# B&R Automation Studio project TestAsProj
Automation Studio 4.12.2.93; Project for testing the OpcUaUnitTesting Python script; technology packages: mappView 5.19.0

## Configuration ARSim

CPU PC_any, AutomationRuntime B4.93, Build 4.1.2, Vc 

### Task classes (Cpu.sw)
```
Cyclic#1 (cycle 10000 us, tolerance 0 us):
  BasicTest <- BasicTest.prg
Cyclic#2 (cycle 20000 us, tolerance 20000 us):
  GetInfo <- GetInfo.prg
Binaries: udbdef, mvLoader, FWRules, OpcUaSrv, TCData, sysconf, Role, User, iomap, ashwd, asfw, arconfig, ashwac
Libraries: arssl, fileio, AsARCfg, runtime, AsBrStr
```

### Hardware
```
PC : PC_any v1.1.1.0 (OrderNumber=PC)
  Connector IF3:
    InternetAddress = 172.27.224.1
  ConfigurationID = TestAsProj_ARSim
  Cyclic1Duration = 10000
  Cyclic1Tolerance = 0
  Cyclic2Duration = 20000
  Cyclic2Tolerance = 20000
  FileDevice1
  FileDeviceName1 = USER
  FileDevicePath1 = USER_PATH
  ActivateOpcUa = 1
  OpcUaInformationModels_PV_Version = 1
```

### Config.mpaudittrail - PC/mappServices/Config.mpaudittrail
```
Element gAuditTrail (Type=mpaudittrail)
  Audit:
    Events:
      [0] = 16
      [1] = 19
    TextSource = TXT
      OutputFormat = MpAudit/Event/Root
    Export:
      Encrypt = FALSE
  Alarms = MpAlarmX
```

### Config_1.mpalarmxcore - PC/mappServices/Config_1.mpalarmxcore
```
Element gAlarmXCore (Type=mpalarmxcore)
```

## Logical view

Binary libraries used (declarations not repeated): operator, runtime, astime, AsIecCon, AsBrStr, AsARCfg

### Global.typ - Global data types
```iecst
TYPE
	GlobalTestStruct : 	STRUCT
		TestUDINT : UDINT;
		TestBOOL : BOOL;
		TestSTRING : STRING[50];
		TestSubStruct : GlobalTestSubStruct;
	END_STRUCT;
	GlobalTestSubStruct : 	STRUCT
		TestREAL : REAL;
		TestLREAL : LREAL;
	END_STRUCT;
END_TYPE
```

### Global.var - Global variables
```iecst
VAR
	gGlobalInt : INT := -100;
	gGlobalUInt : UINT := 100;
	gGlobalString : STRING[50] := 'Test String?!';
	gTestStruct : GlobalTestStruct := (TestUDINT:=45678,TestBOOL:=TRUE,TestSTRING:='Test String 2',TestSubStruct:=(TestREAL:=123.4,TestLREAL:=432.1));
END_VAR
```

### Package Logical/Libraries - Global libraries

- Visualisation Logical/mappView (not shown)

### Program Logical/GetInfo (IEC)

#### Types.typ
```iecst
TYPE
	VisInfo_type : 	STRUCT
		IpAddr : STRING[80];
		NumConnectedClients : USINT;
		IsItFriday : STRING[10];
	END_STRUCT;
	InfoRefreshState_enum :
		(
		INFO_REFRESH_STATE_WAIT,
		INFO_REFRESH_STATE_GET_IP,
		INFO_REFRESH_STATE_GET_DAY,
		INFO_REFRESH_STATE_ERROR
		);
END_TYPE
```

#### Variables.var
```iecst
VAR
	VisInfo : VisInfo_type;
	InfoRefreshState : InfoRefreshState_enum;
	CmdRefreshInfo : BOOL;
	CmdErrorReset : BOOL;
	Error : BOOL;
	DtStruct : DTStructure;
END_VAR
(*Function Blocks*)
VAR
	fb_CfgGetIpAddr : CfgGetIPAddr;
	fb_DTStructureGetTime : DTStructureGetTime;
END_VAR
```

#### Main.st
```iecst
PROGRAM _INIT
    CmdRefreshInfo := TRUE;

END_PROGRAM

PROGRAM _CYCLIC
    CASE InfoRefreshState OF
        INFO_REFRESH_STATE_WAIT:
            IF CmdRefreshInfo THEN
                CmdRefreshInfo := FALSE;
                InfoRefreshState := INFO_REFRESH_STATE_GET_IP;
            END_IF;

        INFO_REFRESH_STATE_GET_IP:
            fb_CfgGetIpAddr.enable := TRUE;
            fb_CfgGetIpAddr.pDevice := ADR('IF3');
            fb_CfgGetIpAddr.pIPAddr := ADR(VisInfo.IpAddr);
            fb_CfgGetIpAddr.Len := SIZEOF(VisInfo.IpAddr);

            IF (fb_CfgGetIpAddr.status <> ERR_FUB_BUSY) AND (fb_CfgGetIpAddr.status <> ERR_FUB_ENABLE_FALSE) THEN
                IF fb_CfgGetIpAddr.status = ERR_OK THEN
                    fb_CfgGetIpAddr.enable := FALSE;
                    InfoRefreshState := INFO_REFRESH_STATE_GET_DAY;
                ELSE
                    Error := TRUE;
                    InfoRefreshState := INFO_REFRESH_STATE_ERROR;
                END_IF;
            END_IF;

        INFO_REFRESH_STATE_GET_DAY:
            brsmemset(ADR(VisInfo.IsItFriday), 0, SIZEOF(VisInfo.IsItFriday));
            brsstrcpy(ADR(VisInfo.IsItFriday), ADR('No :('));

            fb_DTStructureGetTime.enable := TRUE;
            fb_DTStructureGetTime.pDTStructure := ADR(DtStruct);

            IF (fb_DTStructureGetTime.status <> ERR_FUB_BUSY) AND (fb_DTStructureGetTime.status <> ERR_FUB_ENABLE_FALSE) THEN
                IF fb_DTStructureGetTime.status = ERR_OK THEN
                    fb_DTStructureGetTime.enable := FALSE;
                    IF DtStruct.wday = 5 THEN
                        brsmemset(ADR(VisInfo.IsItFriday), 0, SIZEOF(VisInfo.IsItFriday));
                        brsstrcpy(ADR(VisInfo.IsItFriday), ADR('Yes!'));
                    END_IF;
                    InfoRefreshState := INFO_REFRESH_STATE_WAIT;
                ELSE
                    Error := TRUE;
                    InfoRefreshState := INFO_REFRESH_STATE_ERROR;
                END_IF;
            END_IF;

        INFO_REFRESH_STATE_ERROR:
            IF CmdErrorReset THEN
                CmdErrorReset := FALSE;
                Error := FALSE;
                fb_CfgGetIpAddr.enable := FALSE;
                InfoRefreshState := INFO_REFRESH_STATE_WAIT;
            END_IF;

    END_CASE;

    //Call function blocks
    fb_CfgGetIpAddr();
    fb_DTStructureGetTime();
END_PROGRAM
```

### Program Logical/BasicTest (IEC)

#### Variables.var
```iecst
VAR
	TestBOOL : BOOL := TRUE;
	TestDINT : DINT := 65534;
	TestDT : DATE_AND_TIME;
	TestTIME : TIME := T#1d;
	AdditionIn1 : REAL;
	AdditionIn2 : REAL;
	AdditionOut : REAL;
END_VAR
```

#### Main.st
```iecst
PROGRAM _INIT
    gGlobalInt;
    gGlobalUInt;
    gGlobalString;
    gTestStruct;

    TestBOOL;
    TestDINT;
    TestDT;
    TestTIME;

END_PROGRAM

PROGRAM _CYCLIC
	AdditionOut := AdditionIn1 + AdditionIn2;

END_PROGRAM
```

### Program Logical/Alarms

#### Variables.var
```iecst
VAR
	fb_MpAlarmXCore : MpAlarmXCore;
END_VAR
```

#### Main.st
```iecst
PROGRAM _INIT
    fb_MpAlarmXCore.MpLink := ADR(gAlarmXCore);
    fb_MpAlarmXCore.Enable := TRUE;

END_PROGRAM

PROGRAM _CYCLIC
	fb_MpAlarmXCore();

END_PROGRAM

PROGRAM _EXIT
	fb_MpAlarmXCore(Enable := FALSE);

END_PROGRAM
```

### Program Logical/Audit

#### Variables.var
```iecst
VAR
	fb_MpAuditTrail : MpAuditTrail;
END_VAR
```

#### Main.st
```iecst
PROGRAM _INIT
    fb_MpAuditTrail.MpLink := ADR(gAuditTrail);
    fb_MpAuditTrail.Enable := TRUE;
    fb_MpAuditTrail.DeviceName := ADR('FD_Audit');

END_PROGRAM

PROGRAM _CYCLIC
	fb_MpAuditTrail();

END_PROGRAM

PROGRAM _EXIT
	fb_MpAuditTrail(Enable := FALSE);

END_PROGRAM
```

### Program Logical/WaterHeat

#### Main.st
```iecst
PROGRAM _INIT
    // Initial values
    WaterTemperature := BASE_TEMPERATURE;
    WaterLevel := 0.0;

    HeatRate := 0.3;
    CoolRate := 0.1;
    FillRate := 1.0;
    DrainRate := 1.0;

END_PROGRAM

PROGRAM _CYCLIC
	// Heating
    IF HeaterOn THEN
        WaterTemperature := WaterTemperature + (HeatRate/CYCLES_PER_SECOND);
    ELSE
        WaterTemperature := WaterTemperature - (CoolRate/CYCLES_PER_SECOND);
    END_IF;

    IF WaterTemperature > MAX_TEMPERATURE THEN
        WaterTemperature := MAX_TEMPERATURE;
    ELSIF WaterTemperature < BASE_TEMPERATURE THEN
        WaterTemperature := BASE_TEMPERATURE;
    END_IF;

    // Filling and Draining
    IF FillValveOpen THEN
        WaterLevel := WaterLevel + (FillRate/CYCLES_PER_SECOND);
    END_IF;

    IF DrainValveOpen THEN
        WaterLevel := WaterLevel - (DrainRate/CYCLES_PER_SECOND);
    END_IF;

    IF WaterLevel > MAX_LEVEL THEN
        WaterLevel := MAX_LEVEL;
        FillValveOpen := FALSE;
    ELSIF WaterLevel < MIN_LEVEL THEN
        WaterLevel := MIN_LEVEL;
        DrainValveOpen := FALSE;
    END_IF;

END_PROGRAM
```
